// TIA Portal V16 export
// export: Created 2024-12-03T15:41:46.6272737Z, ExportSetting WithReadOnly, DisplayName Totally Integrated Automation Portal, DisplayVersion V16 Update 6, DisplayName TIA Portal Version Control Interface, DisplayVersion V16 Update 2, DisplayName TIA Portal Openness, DisplayVersion V16 Update 6, DisplayName TIA Portal Teamcenter Gateway, DisplayVersion V16, DisplayName SINAMICS Startdrive Advanced, DisplayVersion V16 Update 5, DisplayName SINAMICS Startdrive G130, G150, S120, S150, SINAMICS MV, S210, DisplayVersion V16 Update 5, DisplayName SINAMICS Startdrive G110M, G120, G120C, G120D, G120P, G115D, DisplayVersion V16 Update 5, DisplayName STEP 7 Professional, DisplayVersion V16 Update 6, DisplayName STEP 7 Safety, DisplayVersion V16, DisplayName WinCC Advanced / Unified PC, DisplayVersion V16 Update 6
VAR_GLOBAL   // PLC tag table "10 ConveyLinx"
   I_CON_102 AT %I0.0 : "CLXAiPLC_IN_UDT";
   Q_CON_102 AT %Q0.0 : "CLXAiPLC_OUT_UDT";
   I_CON_103 AT %I64.0 : "CLXAiPLC_IN_UDT";
   Q_CON_103 AT %Q64.0 : "CLXAiPLC_OUT_UDT";
   I_CON_104 AT %I128.0 : "CLXAiPLC_IN_UDT";
   Q_CON_104 AT %Q128.0 : "CLXAiPLC_OUT_UDT";
   I_CON_105 AT %I192.0 : "CLXAiPLC_IN_UDT";
   Q_CON_105 AT %Q192.0 : "CLXAiPLC_OUT_UDT";
   I_CON_106 AT %I256.0 : "CLXAiPLC_IN_UDT";
   Q_CON_106 AT %Q256.0 : "CLXAiPLC_OUT_UDT";
   I_CON_107 AT %I320.0 : "CLXAiPLC_IN_UDT";
   Q_CON_107 AT %Q320.0 : "CLXAiPLC_OUT_UDT";
   I_CON_108 AT %I384.0 : "CLXAiPLC_IN_UDT";
   Q_CON_108 AT %Q384.0 : "CLXAiPLC_OUT_UDT";
   I_CON_109 AT %I448.0 : "CLXAiPLC_IN_UDT";
   Q_CON_109 AT %Q448.0 : "CLXAiPLC_OUT_UDT";
   I_CON_110 AT %I512.0 : "CLXAiPLC_IN_UDT";
   Q_CON_110 AT %Q512.0 : "CLXAiPLC_OUT_UDT";
   I_CON_111 AT %I576.0 : "CLXAiPLC_IN_UDT";
   Q_CON_111 AT %Q576.0 : "CLXAiPLC_OUT_UDT";
   I_CON_112 AT %I640.0 : "CLXAiPLC_IN_UDT";
   Q_CON_112 AT %Q640.0 : "CLXAiPLC_OUT_UDT";
   I_CON_113 AT %I704.0 : "CLXAiPLC_IN_UDT";
   Q_CON_113 AT %Q704.0 : "CLXAiPLC_OUT_UDT";
   I_CON_114 AT %I768.0 : "CLXAiPLC_IN_UDT";
   Q_CON_114 AT %Q768.0 : "CLXAiPLC_OUT_UDT";
   I_CON_115 AT %I832.0 : "CLXAiPLC_IN_UDT";
   Q_CON_115 AT %Q832.0 : "CLXAiPLC_OUT_UDT";
   I_CON_202 AT %I896.0 : "CLXAiPLC_IN_UDT";
   Q_CON_202 AT %Q896.0 : "CLXAiPLC_OUT_UDT";
   I_CON_203 AT %I960.0 : "CLXAiPLC_IN_UDT";
   Q_CON_203 AT %Q960.0 : "CLXAiPLC_OUT_UDT";
   I_CON_301 AT %I1024.0 : "CLXAiPLC_IN_UDT";
   Q_CON_301 AT %Q1024.0 : "CLXAiPLC_OUT_UDT";
   I_CON_302 AT %I1088.0 : "CLXAiPLC_IN_UDT";
   Q_CON_302 AT %Q1088.0 : "CLXAiPLC_OUT_UDT";
   I_CON_303 AT %I1152.0 : "CLXAiPLC_IN_UDT";
   Q_CON_303 AT %Q1152.0 : "CLXAiPLC_OUT_UDT";
   I_CON_304 AT %I1216.0 : "CLXAiPLC_IN_UDT";
   Q_CON_304 AT %Q1216.0 : "CLXAiPLC_OUT_UDT";
   I_CON_305 AT %I1280.0 : "CLXAiPLC_IN_UDT";
   Q_CON_305 AT %Q1280.0 : "CLXAiPLC_OUT_UDT";
   I_CON_201 AT %I1354.0 : "CLXAiPLC_IN_UDT";
   Q_CON_201 AT %Q1352.0 : "CLXAiPLC_OUT_UDT";
END_VAR
